(* IEC 61131-3 sources: HPLC/template/projeto-plc/blocks, 3 files *)

(* ---- 00_FB_InstrumentoAnalogico.st ---- *)
FUNCTION_BLOCK FB_InstrumentoAnalogico
VAR_INPUT
    ValorRaw : INT;
    HabilitaSimulacao : BOOL;
    ValorSimulado : REAL;
    RangeLow : REAL;
    RangeHigh : REAL;
    AlarmeLow : REAL;
    AlarmeHigh : REAL;
END_VAR
VAR_OUTPUT
    ValorEngenharia : REAL;
    ValorFisico : REAL;
    StatusLow : BOOL;
    StatusHigh : BOOL;
    Desconectado : BOOL;
END_VAR

ValorFisico := INT_TO_REAL(ValorRaw) * 20.0 / 32767.0;
Desconectado := (ValorRaw < 0) OR (ValorRaw > 32767);
IF HabilitaSimulacao THEN
    ValorEngenharia := ValorSimulado;
ELSE
    ValorEngenharia := RangeLow + INT_TO_REAL(ValorRaw) * (RangeHigh - RangeLow) / 32767.0;
END_IF;
StatusLow := (ValorEngenharia <= AlarmeLow) AND NOT Desconectado;
StatusHigh := (ValorEngenharia >= AlarmeHigh) AND NOT Desconectado;
END_FUNCTION_BLOCK

(* ---- 10_FB_Motor.st ---- *)
FUNCTION_BLOCK FB_Motor
VAR_INPUT
    ComandoAutomatico : BOOL;
    ComandoManual : BOOL;
    HabilitaManual : BOOL;
    PermiteOperacao : BOOL;
    RetornoLigado : BOOL;
END_VAR
VAR_OUTPUT
    ComandoSaida : BOOL;
    EmOperacao : BOOL;
    Falha : BOOL;
END_VAR

IF HabilitaManual THEN
    ComandoSaida := ComandoManual AND PermiteOperacao;
ELSE
    ComandoSaida := ComandoAutomatico AND PermiteOperacao;
END_IF;
EmOperacao := ComandoSaida AND RetornoLigado;
Falha := ComandoSaida AND NOT RetornoLigado;
END_FUNCTION_BLOCK

(* ---- 20_FB_Valvula.st ---- *)
FUNCTION_BLOCK FB_Valvula
VAR_INPUT
    ComandoAutomatico : BOOL;
    ComandoManual : BOOL;
    HabilitaManual : BOOL;
    PermiteAbrir : BOOL;
    RetornoAberta : BOOL;
    RetornoFechada : BOOL;
END_VAR
VAR_OUTPUT
    ComandoSaida : BOOL;
    Aberta : BOOL;
    Fechada : BOOL;
    Falha : BOOL;
END_VAR

IF HabilitaManual THEN
    ComandoSaida := ComandoManual AND PermiteAbrir;
ELSE
    ComandoSaida := ComandoAutomatico AND PermiteAbrir;
END_IF;
Aberta := RetornoAberta;
Fechada := RetornoFechada;
Falha := RetornoAberta AND RetornoFechada;
END_FUNCTION_BLOCK
